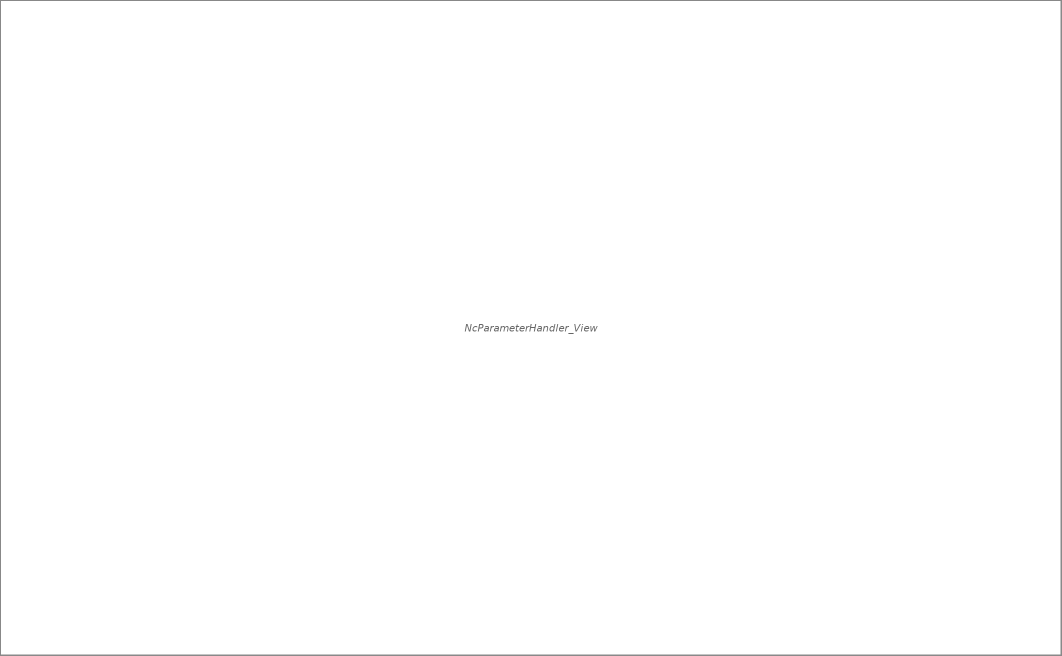
VISUALIZATION View_Test  // 1062x656
    TabControl (0,0 1062x656)
        shows NcParameterHandler_View(DataContent := PRG_TEST.NcPHandler_VM)
        [0]: TabTitle=NC Axis
END_VISUALIZATION

(* stored: Version 1.1.0.1, ProductVersion 3.1.4024.12
   Visu View_Test: Id {868af1aa-845b-06e7-3976-0fc729537f2c} *)
